TEXTLIST KUnLoadMode
  0 = 'Suction'
  1 = 'Position'
   = ''
END_TEXTLIST

(* stored: Version 1.1.0.1, ProductVersion 3.1.4024.11
   TextList KUnLoadMode: Id {cd99a21b-28a6-4469-8024-981d015f0023} *)
